{attribute 'GeneratedUsingTerminal: EP9128-0021-0016'}
{attribute addProperty BoxType "EP9128-0021-0016"}
{attribute addProperty Id "A_0007_EP9128_0021_0017A_0007_EP9128_0021_0017_DAB873EE587A_0004_EP9128_0021_0016_2_EP9128_1021EP9128_AB5A94672"}
{attribute addProperty CRC "1042201659"}
{attribute addProperty Size "589"}
TYPE A_0004_EP9128_0021_0016_3E1EBC3B EXTENDS EP9128_AB5A9467 :
STRUCT
	{attribute addProperty Name "A_0007_EP9128_0021_0017"}
	A_0007_EP9128_0021_0017 : A_0007_EP9128_0021_0017_DAB873EE;
	{attribute addProperty Name "A_0004_EP9128_0021_0016_2_EP9128_1021"}
	A_0004_EP9128_0021_0016_2_EP9128_1021 : EP9128_AB5A9467;
END_STRUCT
END_TYPE

(* stored: Version 1.2.0.0, ProductVersion 3.1.4024.9
   DUT A_0004_EP9128_0021_0016_3E1EBC3B: Id {0bda6bc5-59f8-42f9-833d-496af75c1045} *)
